{attribute addProperty BoxType "EL9222-4433-0018"}
{attribute addProperty Id "OCP_Inputs_ChannelAT %I*ARRAY[0..1] OF OCP_Inputs_Channel_FE08AF3C6480OCP_Outputs_ChannelAT %Q*ARRAY[0..1] OF OCP_Outputs_Channel_F330A9163240WcStateAT %I*WcState_F855686C1620InfoDataAT %I*InfoData_BC63D37F80100"}
{attribute addProperty CRC "901363556"}
{attribute addProperty SizeInBites "192"}
{attribute addProperty SizeInBytes "24"}
TYPE EL9222_39D75EBE :
STRUCT
	{attribute addProperty Name "OCP_Inputs_Channel"}
	OCP_Inputs_Channel : ARRAY[0..1] OF OCP_Inputs_Channel_FE08AF3C;
	{attribute addProperty Name "OCP_Outputs_Channel"}
	OCP_Outputs_Channel : ARRAY[0..1] OF OCP_Outputs_Channel_F330A916;
	{attribute addProperty Name "WcState"}
	WcState : WcState_F855686C;
	{attribute addProperty Name "InfoData"}
	InfoData : InfoData_BC63D37F;
END_STRUCT
END_TYPE

(* stored: Version 1.2.0.0, ProductVersion 3.1.4024.9
   DUT EL9222_39D75EBE: Id {f1b2a98d-fe29-4c70-b49f-bf4babf51944} *)
